// TIA Portal V17 export
// export: Created 2022-12-09T10:51:17.1686495Z, ExportSetting WithDefaults, DisplayName Totally Integrated Automation Portal, DisplayVersion V17 Update 5, DisplayName TIA Portal Openness, DisplayVersion V17 Update 5, DisplayName TIA Portal Version Control Interface, DisplayVersion V17, DisplayName Simotion SCOUT TIA, DisplayVersion 5.4.3.0, DisplayName SINAMICS Startdrive Advanced, DisplayVersion V17 SP1, DisplayName SINAMICS Startdrive G130, G150, S120, S150, SINAMICS MV, S210, DisplayVersion V17 SP1, DisplayName SINAMICS Startdrive G110M, G120, G120C, G120D, G120P, G115D, DisplayVersion V17 SP1, DisplayName STEP 7 Professional, DisplayVersion V17 Update 5, DisplayName STEP 7 Safety, DisplayVersion V17, DisplayName WinCC Advanced, DisplayVersion V17 Update 5
TYPE "NDSN_ST_Ctrl_Sts"
// stored: IsFailsafeCompliant false
   STRUCT
      b_r_SystemReady : Bool;
      b_r_Fault : Bool;
      b_r_Alert : Bool;
      b_r_Stop : Bool;
      b_r_LostCommunication : Bool;
      b_r_TemperatureReady : Bool;
      b_r_HeatersOn : Bool;
      b_r_StandbyOn : Bool;
      b_r_TemperatureAlert : Bool;
      b_r_TemperatureFault : Bool;
      b_r_PumpRunning : Bool;
      b_r_PumpEnabled : Bool;
      b_r_Purging : Bool;
      b_r_TankLevelLow : Bool;
      b_r_TankLevelEmpty : Bool;
      b_r_FillSysAlert : Bool;
      b_r_FillSysFault : Bool;
      b_r_Filling : Bool;
      b_r_LidOpen : Bool;
      b_r_FillLevelSensorCalibrated : Bool;
      b_w_ClearAlertFault : Bool;
      b_w_HeatersOnOff : Bool;
      b_w_StandbyOnOff : Bool;
      b_w_PumpOnOff : Bool;
      b_w_Purge : Bool;
      b_w_ManualFill : Bool;
      b_w_CalibrateEmpty : Bool;
      w_Alarm : Word;
   END_STRUCT;
END_TYPE
